FUNCTION_BLOCK Test_TStreamAdd_Read_ULINT EXTENDS T_UnitTestBase
VAR
    Stream  : T_Stream(StreamLength := 2);
    ArgType : E_ArgTypeId := E_ArgTypeId.Type_ULINT;
END_VAR

{attribute 'analysis' := '-33'} // inhibit unused variable warning
METHOD RunTest

Stream.Init(2);

// add a ULINT...
Stream.SetNextArgTypeId(ArgType);
Stream.Add_ULINT(123456789);

Stream.SetReadPosition(0);

// check next arg type is correct...
AssertEquals_INT(Expected     := ArgType,
                           Actual       := Stream.GetNextArgTypeId(),
                           Message := 'Stream.GetNextArgTypeId()');

// check next value...	
AssertEquals_ULINT(Expected     := 123456789,
                             Actual       := Stream.Read_ULINT(),
                             Message := 'Stream.Read_ULINT()');

// check we are at the end of the stream..							
AssertEquals_UDINT(Expected     := Stream.StreamLength,
                             Actual       := Stream.ReadPosition,
                             Message := 'Stream.ReadPosition');

TestCompleted := TRUE;
END_METHOD

END_FUNCTION_BLOCK

(* stored: Version 1.1.0.1, ProductVersion 3.1.4024.12
   POU Test_TStreamAdd_Read_ULINT: Id {d00d46f5-ceb2-47dd-889b-b54c309f515b}, SpecialFunc None
   Method RunTest: Id {5934fd4f-6c47-4b25-987c-efe3ec001fc4} *)
